Universal Robots PolyScope program: force_torque_tool.urp

Program force_torque_tool (installation=20240827 directory=/programs/Demos/adaptiveGrip createdIn=5.1.0 lastSavedIn=5.15.1 robotSerialNumber=20245500285)
Calibrated DH parameters: a=[0.000097, -0.210459, -0.026602, 0.000137, 0.000078, 0]; d=[0.162601, 254.180657, -54.076236, -199.970743, 0.099615, 0.099684]; alpha=[1.569796, -0.001455, 0.001957, 1.570525, -1.571561, 0]; deltaTheta=[0, -1.053331, 8.839472, -1.50296, 0.000002, 0]
InitVariablesNode
Robot Program (runOnlyOnce=false)
  force_torque := get_tcp_force()
  force_B := p[force_torque[0],force_torque[1],force_torque[2],0,0,0]
  torque_B := p[force_torque[3],force_torque[4],force_torque[5],0,0,0]
  tcp := get_actual_tcp_pose()
  rotation_BT := p[0,0,0,tcp[3],tcp[4],tcp[5]]
  force_T := pose_trans(pose_inv(rotation_BT), force_B)
  torque_T := pose_trans(pose_inv(rotation_BT), torque_B)
  Wait Sleep waitTime=0.01
